# EPICS substitutions: measCompApp/Db/USB1208.substitutions
file "$(MEASCOMP)/db/measCompLongIn.template"
{
pattern
{ R,    MASK,  ADDR}
{Li1, 0xFFFF,     0}
{Li2, 0xFFFF,     1}
}

# This device is a bit confusing.
# For input we read 8-bit word data from ADDR=0,1
# For output we write bit data which must use ADDR=0
file "$(MEASCOMP)/db/measCompBinaryIn.template"
{
pattern
{ R,    MASK,     ADDR}
{ Bi1,  0x01,        0}
{ Bi2,  0x02,        0}
{ Bi3,  0x04,        0}
{ Bi4,  0x08,        0}
{ Bi5,  0x10,        0}
{ Bi6,  0x20,        0}
{ Bi7,  0x40,        0}
{ Bi8,  0x80,        0}
{ Bi9,  0x01,        1}
{Bi10,  0x02,        1}
{Bi11,  0x04,        1}
{Bi12,  0x08,        1}
{Bi13,  0x10,        1}
{Bi14,  0x20,        1}
{Bi15,  0x40,        1}
{Bi16,  0x80,        1}
}

file "$(MEASCOMP)/db/measCompLongOut.template"
{
pattern
{ R,    MASK,    ADDR}
{Lo1, 0xFFFF,       0}
{Lo2, 0xFFFF,       1}
}

file "$(MEASCOMP)/db/measCompBinaryOut.template"
{
pattern
{  R,    MASK,     ADDR}
{ Bo1,   0x01,        0}
{ Bo2,   0x02,        0}
{ Bo3,   0x04,        0}
{ Bo4,   0x08,        0}
{ Bo5,   0x10,        0}
{ Bo6,   0x20,        0}
{ Bo7,   0x40,        0}
{ Bo8,   0x80,        0}
{ Bo9,   0x10,        1}
{Bo10,   0x20,        1}
{Bo11,   0x40,        1}
{Bo12,   0x80,        1}
{Bo13,   0x10,        1}
{Bo14,   0x20,        1}
{Bo15,   0x40,        1}
{Bo16,   0x80,        1}
}

# Direction bits on binary I/O
#  VAL 0=input, 1=output
file "$(MEASCOMP)/db/measCompBinaryDir.template"
{
pattern
{  R,   MASK,  VAL,    ADDR}
{Bd1, 0xFFFF,    0,       0}
{Bd2, 0xFFFF,    0,       1}
}

file "$(MEASCOMP)/db/measCompCounter.template"
{
pattern
{       R,     ADDR}
{Counter1,        0}
}

# Analog input mode
file "$(MEASCOMP)/db/measCompAnalogInMode.template"
{
pattern
{  R,       ADDR,   MODE}
{AiMode,       0,      0}
}

# Analog inputs
file "$(MEASCOMP)/db/measCompAnalogIn.template"
{
pattern
{  R,  ADDR,  EGUL, LOPR, EGUF, HOPR, RANGE,       SCAN, PREC}
{ Ai1,     0,  -10., -10.,  10.,  10.,    1,  "1 second",   4}
{ Ai2,     1,  -10., -10.,  10.,  10.,    1,  "1 second",   4}
{ Ai3,     2,   -5.,  -5.,   5.,   5.,    2,  "1 second",   4}
{ Ai4,     3,   -5.,  -5.,   5.,   5.,    2,  "1 second",   4}
}

# Analog outputs
file "$(MEASCOMP)/db/measCompAnalogOut.template"
{
pattern
{  R, VAL,   ADDR,  EGUL, DRVL, LOPR, EGUF, DRVH, HOPR, PREC}
{Ao1,   0,      0,    0,    0,   0,    5,    5,     5,    4}
{Ao2,   0,      1,    0,    0,   0,    5,    5,     5,    4}
}
